{attribute 'qualified_only'}
{attribute 'strict'}
TYPE eTcoSequencerTests :
(
	none	:= -1,
	CallSequencerBodiesOnly	:= 100,
	RestoreSequencers,
	NumberOfStepsCount := 500,
	ExecutionInOnePLCcycle,
	OnStepCompleted,
	OnSequenceCompleted,
	RestoreChildBetweenSteps,
	OnStateChangeWithRestoreCallInside,
	MinStepId,
	MaxStepId,
	RequestStepToFirstStepWithStepId0,
	RequestStep,
	CheckStepIdUniqueness,
	RestoreAlreadyCheckedSequence:=512,
	NotUniqueStepId,
	AfterErrorRestore := 516,
	ChangeStepIdDuringExecution := 520,
	CommentOutPartOfRunningSequencer := 524,
	UncommentPartOfRunningSequencer:=526,
	OpenCloseSequence := 530,
	RequestStepFromLowerToHigher := 541,
	RequestStepFromHigherToLower:=542,
	RequestStepToNotExistingStep:=544,
	RequestStepWhilePreviousRequestStepHasNotBeenYetProcessed :=547,
	DisableStepEnabledAndActiveInPreviousPLCcycle := 551,
	RequestStepCallingCyclically :=560,
	SetStepMode := 570,
	StepMode :=580,
	InvalidMode :=582,
	StepInError := 583,
	CheckStepIdUniquenessStepMode :=590,
	ResetSequenceInStepMode,
	NotUniqueStepIdInStep,
	ResetInStepModeAfterNotUniqueStepIdError,
	AfterErrorResetInStepMode,
	PrepareForInvalidMode,
	InvalidSequencerMode,
	PrepareForStepInError,
	StepInError_1,
	StepModeFirstCycle := 610,
	StepModeStepIn_1,
	StepModeChangeStepIdDuringExecution,
	StepModeRestoreAfterChangeStepIdDuringExecutionError,
	StepModePrepareSequenceBeforeChangeOrderTest,
	StepModeChangeStepOrder,
	StepModeRestoreAfterChangeStepError,
	StepModePrepareSequenceBeforeCommentOutTest,
	StepModeCommentOutTest,
	StepModeRestoreSequenceAfterCommentOutError,
	StepModePrepareSequenceBeforeUncommentTest,
	StepModeUncommentTest,
	StepModePrepareForRequestStepFromLowerToHigher :=630,
	StepModeRequestStepFromLowerToHigher,
	StepModePrepareForRequestStepFromHigherToLower,
	StepModeRequestStepFromHigherToLowerTriggered,
	StepModeRequestStepFromHigherToLowerExecuted,
	StepModeRequestStepToNotExistingStepFirstCycle,
	StepModeRequestStepToNotExistingStepSecondCycle,
	StepModeRequestStepToNotExistingStepThirdCycle,
	StepModeRestoreAfterRequestStepToNotExistingStepError,
	StepModeRequestStepWhilePreviousRequestStepHasnotBeenYetProcessed:=640,
	StepModePrepareForDisableStepTestFirstCycle,
	StepModePrepareForDisableStepTestNext2Cycles,
	StepModePrepareForDisabledStepTest,
	StepModeStepInCallOnDisabledStep,
	StepModeStepInAfterStepInCallOnDisabledStep,
	StepModePrepareForStepForwardBackwardTestFirstCycle:=670,
	StepModePrepareForStepForwardBackwardTestSecondCycle,
	StepModeStepForward_1,
	StepModeRequestStepToTheLastStepOfTheSequence,
	StepModeStepForward_2,
	StepModeStepBackward_1,
	StepModeRequestBeforeFirstStepOfTheSequence,
	StepModeStepBackward_2,
	StepModeStepBackward_3,
	StepModePrepareForStepInTest := 680,
	StepModeStepIn_2,
	StepModeStepInIntoTheStepInsideWhichRequestStepToTheLastStepOfTheSequence,
	StepModeStepInAfterRequestStepToTheLastStepOfTheSequenceWasCalled,
	StepModeStepInFromLastStepOfTheSequence,
	PrepareSequenceBeforeSwitchStepModeOnDuringStepExecution := 690,
	SwitchStepModeOnDuringStepExecution,
	SwitchStepModePrepareForStepForwardFromRunningStep,
	SwitchStepModeStepForwardFromRunningStep,
	SwitchStepModePrepareForStepBackwardFromRunningStep,
	SwitchStepModeStepBackwardFromRunningStep,
	SwitchStepModeStepOffFromReadyToRun,
	SwitchStepModeStepOnFromRunning,
	SwitchStepModeStepOffFromRunning,
	OnStateChangeWhenChangingModes	
);
END_TYPE

(* stored: Version 1.1.0.1, ProductVersion 3.1.4024.9
   DUT eTcoSequencerTests: Id {e151dbc6-3491-0a9b-19b3-6a566e0dfd83} *)
